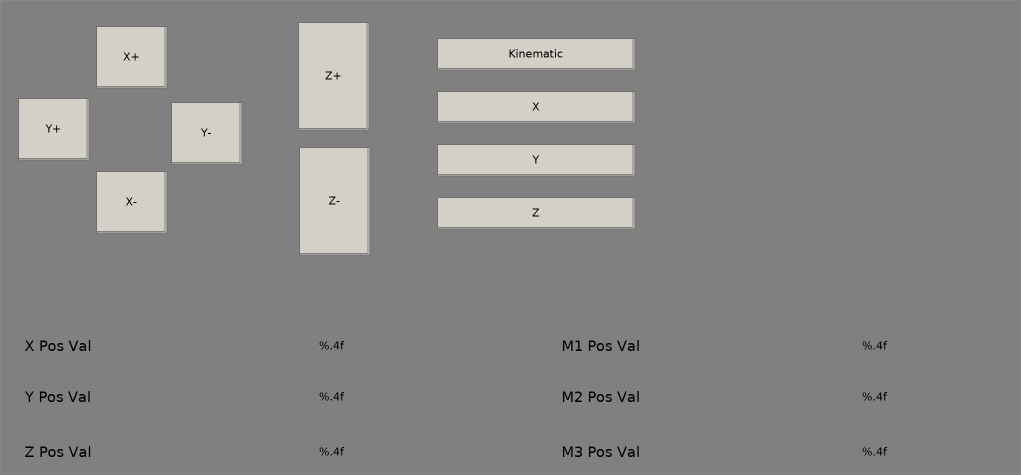
VISUALIZATION Visualization_1  // 1021x475
    Rectangle (187,334 289x24), "%.4f", text variable: GVL_Axis.AxisX.NcToPlc.ActPos
    Rectangle (187,385 289x24), "%.4f", text variable: GVL_Axis.AxisY.NcToPlc.ActPos
    Rectangle (187,440 289x24), "%.4f", text variable: GVL_Axis.AxisZ.NcToPlc.ActPos
    Label (10,325 96x42), "X Pos Val"
    Label (10,376 96x42), "Y Pos Val"
    Label (10,431 96x42), "Z Pos Val"
    Rectangle (730,334 289x24), "%.4f", text variable: GVL_Axis.AxisM1_B.NcToPlc.ActPos
    Rectangle (730,385 289x24), "%.4f", text variable: GVL_Axis.AxisM2_C.NcToPlc.ActPos
    Rectangle (730,440 289x24), "%.4f", text variable: GVL_Axis.AxisM3_A.NcToPlc.ActPos
    Label (553,325 96x42), "M1 Pos Val"
    Label (553,376 96x42), "M2 Pos Val"
    Label (553,431 96x42), "M3 Pos Val"
    Button (437,91 198x32), "X"
        OnMouseClick: toggle stAxisX.In.xMove
    Button (437,144 198x32), "Y"
        OnMouseClick: toggle stAxisY.In.xMove
    Button (437,197 198x32), "Z"
        OnMouseClick: toggle stAxisZ.In.xMove
    Button (437,38 198x32), "Kinematic"
        OnMouseClick: toggle PRG_Kinematic.bExecuteKinConfigGroup
    Button (96,26 71x62), "X+"
        tap POU_VisButton.xUp
    Button (96,171 71x62), "X-"
        tap POU_VisButton.xDown
    Button (171,102 71x62), "Y-"
        tap POU_VisButton.yDown
    Button (18,98 71x62), "Y+"
        tap POU_VisButton.yUp
    Button (298,22 71x108), "Z+"
        tap POU_VisButton.zuP
    Button (299,147 71x108), "Z-"
        tap POU_VisButton.zDown
END_VISUALIZATION

(* stored: Version 1.1.0.1, ProductVersion 3.1.4024.0
   Visu Visualization_1: Id {6c15c763-3d49-40fc-9046-7619740d9357} *)
